{attribute 'qualified_only'}
{attribute 'strict'}
{attribute 'to_string'}
TYPE States :
(
    OFF := 0,
    ERROR := 1,
    READY := 2,
    RUNNINGv := 3,
    BACKLASH := 4,
    UNDEFINED := 5
);
END_TYPE

(* stored: Version 1.1.0.1
   DUT E_MachineState: Id {3dcb30fc-2b5a-4892-8669-8b9797b6ff58} *)
